FUNCTION_BLOCK FB_Estacion
VAR_INPUT
    EstadoPausa: BOOL;
    EstadoReinicia: BOOL;
    CiclosSolicitados: UINT := 0;
	CiclosRechazados: UINT := 0;
    
    Tcheck: TIME := T#1S;
    Treset: TIME := T#1S;
    Tdesplazador: TIME := T#1S;
	Tcinta: TIME := T#0.5S;
END_VAR
VAR_OUTPUT
    CondicionInicial: BOOL := TRUE;
    CiclosPendientes: UINT;
    CiclosAceptados: UINT;
    PaleCodigo: BYTE;
	pieza_ok: BOOL;
    
    // Entradas comunes
	Base_en_alimentador AT %I*: BOOL;
    Pulsador_parada_emergencia AT %I*: BOOL;
    Selector_modo_manual AT %I*: BOOL;
    Pulsador_marcha AT %I*: BOOL;
    Pulsador_parada_NC AT %I*: BOOL := TRUE; // Contacto normalmente cerrado
    EstacionConectada AT %I*: BOOL := TRUE;
    Detector_presion AT %I*: BOOL := TRUE;

    Presencia_pale AT %I*: BOOL;
    Codigo_pale_bit_0 AT %I*: BOOL; //no lo usamos
    Codigo_pale_bit_1 AT %I*: BOOL; //no lo usamos
    Codigo_pale_bit_2 AT %I*: BOOL; //no lo usamos

    // Entradas espeficicas
    //Terminal 6
	Horizontal_descargador_detras AT %I*: BOOL;
	Horizontal_descargador_delante AT %I*: BOOL;
	Vertical_descargador_arriba AT %I*: BOOL;
	Vertical_descargador_abajo AT %I*: BOOL;
	Verificador_arriba AT %I*: BOOL;
	Verificador_abajo AT %I*: BOOL;
	Desplazador_detras AT %I*: BOOL;
	Desplazador_delante AT %I*: BOOL;
	Alimentador_detras AT %I*: BOOL;
	
	
	//Terminal 7
	Alimentador_delante AT %I*: BOOL;
	Vacio_obtenido_vacuostato_descargador AT %I*: BOOL;

END_VAR
VAR
    // Bloques funcionales
    Coordinador: FB_Coordinador_SFC;
	ChequeaMaterial: FB_CheckMaterial_SFC;
	AlimentadorVerificadorDesplazador: FB_AlimentadorVerificadorDesplazador_SFC;
    SituarPale: FB_SituarPale_SFC;
	ResetDescargador: FB_ResetDescargador_SFC;
    Descargador: FB_Descargador_SFC;
    Rechazador: FB_Rechazador_SFC;
    TransferirPale: FB_TransferirPale_SFC;
    
    // Salidas comunes
    Desconecta_parte_operativa AT %Q*: BOOL;
    Lampara_falta_material AT %Q*: BOOL;
    Lampara_marcha AT %Q*: BOOL;
    Lampara_alarma AT %Q*: BOOL;

    Activa_marcha_motor_cinta AT %Q*: BOOL;
    Invierte_marcha_motor_cinta AT %Q*: BOOL;
    Retenedor_pale_baja AT %Q*: BOOL;
    Separador_pale_sube AT %Q*: BOOL;
    
    //Terminal 8
	Descargador_adelante AT %Q*: BOOL;
	Descargador_atras AT %Q*: BOOL;
	Descargador_baja AT %Q*: BOOL;
	Rechazador_adelante AT %Q*: BOOL;
	Verificador_baja AT %Q*: BOOL;
	Desplazador_adelante AT %Q*: BOOL;
	Alimentador_adelante AT %Q*: BOOL;
	Eyector_succiona AT %Q*: BOOL;
END_VAR

// Modo Automático
IF NOT Selector_Modo_Manual THEN
	
	// Bloques Funcionales
	Coordinador(
		CiclosRechazados := CiclosRechazados,
		CiclosPendientes := CiclosPendientes,
		CiclosAceptados := CiclosAceptados,
		CiclosSolicitados := CiclosSolicitados,
		SFCPause := NOT EstadoReinicia AND EstadoPausa,
        SFCReset := EstadoReinicia,
		Ack := TRUE,
        Execute := Pulsador_marcha AND (CiclosSolicitados > 0),
		PaleSituado := SituarPale.Done,
		HayMaterial := ChequeaMaterial.Done,
		Verificado := AlimentadorVerificadorDesplazador.Done,
		DescargadorReseteado := ResetDescargador.Done,
        Rechazado := Rechazador.Done,
		BaseCargada := Descargador.Done,
		PaleTransferido := TransferirPale.Done,
		Base_en_alimentador := Base_en_alimentador,
		pieza_ok := pieza_ok
		
	);
	
	SituarPale(

		SFCPause := NOT EstadoReinicia AND EstadoPausa,
        SFCReset := EstadoReinicia,
        Ack := NOT Coordinador.SituaPale,
        Execute := Coordinador.SituaPale,
        Tcinta := Tcinta,
        Presencia_pale := Presencia_pale,
       	//Codigo_pale_bit_0 := Codigo_pale_bit_0,
        //Codigo_pale_bit_1 := Codigo_pale_bit_1,
        //Codigo_pale_bit_2 := Codigo_pale_bit_2

	);
	
	ChequeaMaterial(
		Ack := NOT Coordinador.ChequeaMaterial,
		SFCPause := NOT EstadoReinicia AND EstadoPausa,
        SFCReset := EstadoReinicia,
		Execute := Coordinador.ChequeaMaterial,
		Base_en_Alimentador := Base_en_alimentador,
		Pulsador_marcha := Pulsador_marcha
	);
	
	AlimentadorVerificadorDesplazador(
		
		Ack := NOT Coordinador.VerificaBase,
		Tcheck := Tcheck,
		SFCPause := NOT EstadoReinicia AND EstadoPausa,
        SFCReset := EstadoReinicia,
		Execute := Coordinador.VerificaBase,
		Alimentador_delante := Alimentador_delante,
		Alimentador_detras := Alimentador_detras,
		Verificador_arriba := Verificador_arriba ,
		Verificador_abajo := Verificador_abajo,
		Desplazador_delante := Desplazador_delante,
		Desplazador_detras := Desplazador_detras, 
		
	);
	
	ResetDescargador(

		Ack := NOT Coordinador.ResetDescargador,
		SFCPause := NOT EstadoReinicia AND EstadoPausa,
        SFCReset := EstadoReinicia,
		Execute := Coordinador.ResetDescargador,
		Horizontal_descargador_detras := Horizontal_descargador_detras,
		Vertical_descargador_arriba := Vertical_descargador_arriba
	);
	
	Descargador(
		
		Ack := NOT Coordinador.CargaBase,
		SFCPause := NOT EstadoReinicia AND EstadoPausa,
        SFCReset := EstadoReinicia,
		Execute := Coordinador.CargaBase,
		Horizontal_descargador_detras := Horizontal_descargador_detras,
		Vertical_descargador_abajo := Vertical_descargador_abajo,
		Vacio_obtenido_vacuostato_descargador := Vacio_obtenido_vacuostato_descargador ,
		Vertical_descargador_arriba := Vertical_descargador_arriba ,
		Horizontal_descargador_delante := Horizontal_descargador_delante ,
	
	);	
		
	Rechazador(
		
		Ack := NOT Coordinador.RechazaBase,
		SFCPause := NOT EstadoReinicia AND EstadoPausa,
        SFCReset := EstadoReinicia,
		Execute := Coordinador.RechazaBase,
		Verificador_abajo := Verificador_abajo
		
	);
	
	TransferirPale(
	
		Ack := NOT Coordinador.TransfierePale,
		SFCPause := NOT EstadoReinicia AND EstadoPausa,
        SFCReset := EstadoReinicia,
		Execute := Coordinador.TransfierePale,

	);
	
	//Acciones Comunes
	Lampara_falta_material := Coordinador.Lampara_falta_material;
	Activa_marcha_motor_cinta := SituarPale.Activa_marcha_motor_cinta OR TransferirPale.Activa_marcha_motor_cinta;
	//CheckMaterial
	Lampara_alarma := ChequeaMaterial.LamparaAlarma;
	Lampara_falta_material := ChequeaMaterial.Lampara_falta_material;
	//TranferirPale
	 Retenedor_pale_baja := TransferirPale.Retenedor_pale_baja;
	 Separador_pale_sube := TransferirPale.Separador_pale_sube;
	//AlimentadorVerificadorDesplazador
	Alimentador_adelante := AlimentadorVerificadorDesplazador.Alimentador_adelante;
	Verificador_baja := AlimentadorVerificadorDesplazador.Verificador_baja;
	Desplazador_adelante := AlimentadorVerificadorDesplazador.Desplazador_adelante;
	pieza_ok := AlimentadorVerificadorDesplazador.pieza_ok;
	//Descargador
	Eyector_succiona := Descargador.Eyector_succiona;
	Descargador_adelante := Descargador.Descargador_adelante;
	Descargador_atras := Descargador.Descargador_atras OR ResetDescargador.Descargador_atras;
	Descargador_baja := Descargador.Descargador_baja;
	//Rechazador
	Rechazador_adelante := Rechazador.Rechazador_adelante;
	
	IF NOT EstadoPausa THEN
	
		EstadoPausa := not Pulsador_parada_NC;
	
	ELSE
	
		EstadoPausa := NOT Pulsador_marcha;
	
	END_IF

END_IF

END_FUNCTION_BLOCK

(* stored: Version 1.1.0.1, ProductVersion 3.1.4024.12
   POU FB_Estacion: Id {b931997a-e702-4e5f-99bc-19509e72a06d}, SpecialFunc None *)
